LIN {X 0,Y 60.656,Z 289.694,A -85,B 0,C 180,E1 -29046.277,E2 -29046.277} C_VEL
LIN {X 0,Y 62.988,Z 293.733,A -85,B 0,C 180,E1 -29049.53,E2 -29049.53} C_VEL
LIN {X 0,Y 65.947,Z 299.714,A -85,B 0,C 180,E1 -29053.566,E2 -29053.566} C_VEL
LIN {X 0,Y 68.573,Z 306.402,A -85,B 0,C 180,E1 -29057.552,E2 -29057.552} C_VEL
LIN {X 0,Y 68.698,Z 316.329,A -85,B 0,C 180,E1 -29061.954,E2 -29061.954} C_VEL
LIN {X 0,Y 68.38,Z 324.783,A -85,B 0,C 180,E1 -29066.316,E2 -29066.316} C_VEL
LIN {X 0,Y 68.151,Z 327.44,A -85,B 0,C 180,E1 -29067.783,E2 -29067.783} C_VEL
LIN {X 0,Y 64.616,Z 337.01,A -85,B 0,C 180,E1 -29073.116,E2 -29073.116} C_VEL
LIN {X 0,Y 63.028,Z 340.879,A -85,B 0,C 180,E1 -29075.888,E2 -29075.888} C_VEL
LIN {X 0,Y 60.689,Z 345.121,A -85,B 0,C 180,E1 -29079.055,E2 -29079.055} C_VEL
LIN {X 0,Y 55.431,Z 351.353,A -85,B 0,C 180,E1 -29084.685,E2 -29084.685} C_VEL
LIN {X 0,Y 50.566,Z 356.775,A -85,B 0,C 180,E1 -29092.091,E2 -29092.091} C_VEL
LIN {X 0,Y 49.027,Z 359.751,A -85,B 0,C 180,E1 -29097.765,E2 -29097.765} C_VEL
LIN {X 0,Y 48.568,Z 364.973,A -85,B 0,C 180,E1 -29109.693,E2 -29109.693} C_VEL
LIN {X 0,Y 49.872,Z 368.756,A -85,B 0,C 180,E1 -29120.809,E2 -29120.809} C_VEL
LIN {X 0,Y 51.424,Z 370.545,A -85,B 0,C 180,E1 -29126.86,E2 -29126.86} C_VEL
LIN {X 0,Y 56.208,Z 373.025,A -85,B 0,C 180,E1 -29137.968,E2 -29137.968} C_VEL
LIN {X 0,Y 62.698,Z 374.277,A -85,B 0,C 180,E1 -29147.044,E2 -29147.044} C_VEL
LIN {X 0,Y 70.609,Z 374.345,A -85,B 0,C 180,E1 -29154.464,E2 -29154.464} C_VEL
LIN {X 0,Y 78.89,Z 373.239,A -85,B 0,C 180,E1 -29159.999,E2 -29159.999} C_VEL
LIN {X 0,Y 88.109,Z 370.772,A -85,B 0,C 180,E1 -29164.575,E2 -29164.575} C_VEL
LIN {X 0,Y 94.619,Z 368.411,A -85,B 0,C 180,E1 -29167.103,E2 -29167.103} C_VEL
LIN {X 0,Y 97.441,Z 367.133,A -85,B 0,C 180,E1 -29168.293,E2 -29168.293} C_VEL
LIN {X 0,Y 98.808,Z 366.47,A -85,B 0,C 180,E1 -29172.32,E2 -29172.32} C_VEL
LIN {X 0,Y 99.22,Z 366.449,A -85,B 0,C 180,E1 -29176.459,E2 -29176.459} C_VEL
LIN {X 0,Y 99.233,Z 366.885,A -85,B 0,C 180,E1 -29180.739,E2 -29180.739} C_VEL
LIN {X 0,Y 99.149,Z 367.25,A -85,B 0,C 180,E1 -29182.858,E2 -29182.858} C_VEL
LIN {X 0,Y 98.38,Z 367.841,A -85,B 0,C 180,E1 -29184.381,E2 -29184.381} C_VEL
LIN {X 0,Y 90.661,Z 371.366,A -85,B 0,C 180,E1 -29186.942,E2 -29186.942} C_VEL
LIN {X 0,Y 81.683,Z 374.499,A -85,B 0,C 180,E1 -29190.64,E2 -29190.64} C_VEL
LIN {X 0,Y 76.041,Z 376.045,A -85,B 0,C 180,E1 -29193.715,E2 -29193.715} C_VEL
LIN {X 0,Y 70.723,Z 377.095,A -85,B 0,C 180,E1 -29197.346,E2 -29197.346} C_VEL
LIN {X 0,Y 61.158,Z 377.8,A -85,B 0,C 180,E1 -29206.411,E2 -29206.411} C_VEL
LIN {X 0,Y 57.103,Z 377.566,A -85,B 0,C 180,E1 -29212.021,E2 -29212.021} C_VEL
LIN {X 0,Y 53.866,Z 376.846,A -85,B 0,C 180,E1 -29218.542,E2 -29218.542} C_VEL
LIN {X 0,Y 51.484,Z 375.644,A -85,B 0,C 180,E1 -29225.826,E2 -29225.826} C_VEL
LIN {X 0,Y 49.582,Z 373.048,A -85,B 0,C 180,E1 -29237.726,E2 -29237.726} C_VEL
LIN {X 0,Y 49.718,Z 369.258,A -85,B 0,C 180,E1 -29250.001,E2 -29250.001} C_VEL
LIN {X 0,Y 50.679,Z 363.659,A -85,B 0,C 180,E1 -29262.082,E2 -29262.082} C_VEL
LIN {X 0,Y 52.64,Z 359.148,A -85,B 0,C 180,E1 -29269.5,E2 -29269.5} C_VEL
LIN {X 0,Y 55.776,Z 353.792,A -85,B 0,C 180,E1 -29276.17,E2 -29276.17} C_VEL
LIN {X 0,Y 60.052,Z 347.523,A -85,B 0,C 180,E1 -29281.78,E2 -29281.78} C_VEL
LIN {X 0,Y 64.173,Z 342.283,A -85,B 0,C 180,E1 -29285.098,E2 -29285.098} C_VEL
LIN {X 0,Y 68.246,Z 337.731,A -85,B 0,C 180,E1 -29286.999,E2 -29286.999} C_VEL
LIN {X 0,Y 73.162,Z 342.61,A -85,B 0,C 180,E1 -29294.895,E2 -29294.895} C_VEL
LIN {X 0,Y 72.154,Z 341.482,A -85,B 0,C 180,E1 -29297.015,E2 -29297.015} C_VEL
LIN {X 0,Y 65.005,Z 332.075,A -85,B 0,C 180,E1 -29307.278,E2 -29307.278} C_VEL
LIN {X 0,Y 60.672,Z 322.126,A -85,B 0,C 180,E1 -29317.929,E2 -29317.929} C_VEL
LIN {X 0,Y 58.653,Z 313.599,A -85,B 0,C 180,E1 -29326.135,E2 -29326.135} C_VEL
LIN {X 0,Y 57.356,Z 304.126,A -85,B 0,C 180,E1 -29333.846,E2 -29333.846} C_VEL
LIN {X 0,Y 56.745,Z 292.437,A -85,B 0,C 180,E1 -29341.777,E2 -29341.777} C_VEL
LIN {X 0,Y 56.696,Z 289.467,A -85,B 0,C 180,E1 -29343.558,E2 -29343.558} C_VEL
LIN {X 0,Y 55.101,Z 283.817,A -85,B 0,C 180,E1 -29345.813,E2 -29345.813} C_VEL
LIN {X 0,Y 51.561,Z 285.724,A -85,B 0,C 180,E1 -29373.041,E2 -29373.041} C_VEL
LIN {X 0,Y 52.226,Z 286.714,A -85,B 0,C 180,E1 -29382.289,E2 -29382.289} C_VEL
LIN {X 0,Y 52.707,Z 287.689,A -85,B 0,C 180,E1 -29388.185,E2 -29388.185} C_VEL
LIN {X 0,Y 53.227,Z 289.168,A -85,B 0,C 180,E1 -29394.871,E2 -29394.871} C_VEL
LIN {X 0,Y 53.44,Z 290.095,A -85,B 0,C 180,E1 -29397.987,E2 -29397.987} C_VEL
LIN {X 0,Y 56.844,Z 295.639,A -85,B 0,C 180,E1 -29404.195,E2 -29404.195} C_VEL
LIN {X 0,Y 59.186,Z 300.064,A -85,B 0,C 180,E1 -29408.171,E2 -29408.171} C_VEL
LIN {X 0,Y 61.616,Z 305.81,A -85,B 0,C 180,E1 -29412.574,E2 -29412.574} C_VEL
LIN {X 0,Y 62.723,Z 310.076,A -85,B 0,C 180,E1 -29415.395,E2 -29415.395} C_VEL
LIN {X 0,Y 62.547,Z 317.346,A -85,B 0,C 180,E1 -29418.982,E2 -29418.982} C_VEL
LIN {X 0,Y 62,Z 325.309,A -85,B 0,C 180,E1 -29423.49,E2 -29423.49} C_VEL
LIN {X 0,Y 61.705,Z 327.967,A -85,B 0,C 180,E1 -29425.099,E2 -29425.099} C_VEL
LIN {X 0,Y 57.658,Z 338.002,A -85,B 0,C 180,E1 -29431.271,E2 -29431.271} C_VEL
LIN {X 0,Y 54.497,Z 345.164,A -85,B 0,C 180,E1 -29437.408,E2 -29437.408} C_VEL
LIN {X 0,Y 52.168,Z 350.731,A -85,B 0,C 180,E1 -29443.635,E2 -29443.635} C_VEL
LIN {X 0,Y 49.771,Z 356.978,A -85,B 0,C 180,E1 -29452.848,E2 -29452.848} C_VEL
LIN {X 0,Y 49.027,Z 359.751,A -85,B 0,C 180,E1 -29457.765,E2 -29457.765} C_VEL
LIN {X 0,Y 47.9,Z 362.53,A -85,B 0,C 180,E1 -29463.819,E2 -29463.819} C_VEL
LIN {X 0,Y 45.359,Z 366.458,A -85,B 0,C 180,E1 -29474.592,E2 -29474.592} C_VEL
LIN {X 0,Y 44.558,Z 369.668,A -85,B 0,C 180,E1 -29486.581,E2 -29486.581} C_VEL
LIN {X 0,Y 46.096,Z 371.224,A -85,B 0,C 180,E1 -29493.552,E2 -29493.552} C_VEL
LIN {X 0,Y 51.558,Z 373.469,A -85,B 0,C 180,E1 -29504.179,E2 -29504.179} C_VEL
LIN {X 0,Y 59.02,Z 374.707,A -85,B 0,C 180,E1 -29513.16,E2 -29513.16} C_VEL
LIN {X 0,Y 67.483,Z 374.779,A -85,B 0,C 180,E1 -29519.999,E2 -29519.999} C_VEL
LIN {X 0,Y 77.69,Z 373.447,A -85,B 0,C 180,E1 -29525.689,E2 -29525.689} C_VEL
LIN {X 0,Y 86.636,Z 371.138,A -85,B 0,C 180,E1 -29529.337,E2 -29529.337} C_VEL
LIN {X 0,Y 91.606,Z 369.51,A -85,B 0,C 180,E1 -29531.057,E2 -29531.057} C_VEL
LIN {X 0,Y 92.332,Z 369.276,A -85,B 0,C 180,E1 -29533.2,E2 -29533.2} C_VEL
LIN {X 0,Y 92.644,Z 369.375,A -85,B 0,C 180,E1 -29537.664,E2 -29537.664} C_VEL
LIN {X 0,Y 92.666,Z 369.734,A -85,B 0,C 180,E1 -29541.079,E2 -29541.079} C_VEL
LIN {X 0,Y 90.886,Z 370.534,A -85,B 0,C 180,E1 -29541.886,E2 -29541.886} C_VEL
LIN {X 0,Y 84.501,Z 372.83,A -85,B 0,C 180,E1 -29543.813,E2 -29543.813} C_VEL
LIN {X 0,Y 78.302,Z 374.597,A -85,B 0,C 180,E1 -29546.164,E2 -29546.164} C_VEL
LIN {X 0,Y 71.767,Z 376.041,A -85,B 0,C 180,E1 -29549.316,E2 -29549.316} C_VEL
LIN {X 0,Y 66.637,Z 376.892,A -85,B 0,C 180,E1 -29552.465,E2 -29552.465} C_VEL
LIN {X 0,Y 61.218,Z 377.348,A -85,B 0,C 180,E1 -29556.525,E2 -29556.525} C_VEL
LIN {X 0,Y 51.689,Z 376.906,A -85,B 0,C 180,E1 -29567.171,E2 -29567.171} C_VEL
LIN {X 0,Y 47.955,Z 376.122,A -85,B 0,C 180,E1 -29574.113,E2 -29574.113} C_VEL
LIN {X 0,Y 45.12,Z 374.817,A -85,B 0,C 180,E1 -29582.143,E2 -29582.143} C_VEL
LIN {X 0,Y 42.726,Z 372.012,A -85,B 0,C 180,E1 -29595.717,E2 -29595.717} C_VEL
LIN {X 0,Y 42.728,Z 367.921,A -85,B 0,C 180,E1 -29610.002,E2 -29610.002} C_VEL
LIN {X 0,Y 43.489,Z 363.217,A -85,B 0,C 180,E1 -29621.656,E2 -29621.656} C_VEL
LIN {X 0,Y 45.489,Z 358.662,A -85,B 0,C 180,E1 -29630.344,E2 -29630.344} C_VEL
LIN {X 0,Y 48.748,Z 353.283,A -85,B 0,C 180,E1 -29637.942,E2 -29637.942} C_VEL
LIN {X 0,Y 53.154,Z 346.965,A -85,B 0,C 180,E1 -29644.191,E2 -29644.191} C_VEL
LIN {X 0,Y 57.268,Z 341.647,A -85,B 0,C 180,E1 -29647.852,E2 -29647.852} C_VEL
LIN {X 0,Y 63.326,Z 334.785,A -85,B 0,C 180,E1 -29650.695,E2 -29650.695} C_VEL
LIN {X 0,Y 64.269,Z 333.998,A -85,B 0,C 180,E1 -29651.006,E2 -29651.006} C_VEL
LIN {X 0,Y 65.947,Z 335.721,A -85,B 0,C 180,E1 -29653.846,E2 -29653.846} C_VEL
LIN {X 0,Y 65.682,Z 335.325,A -85,B 0,C 180,E1 -29655.933,E2 -29655.933} C_VEL
LIN {X 0,Y 59.31,Z 326.435,A -85,B 0,C 180,E1 -29665.729,E2 -29665.729} C_VEL
LIN {X 0,Y 54.783,Z 315.648,A -85,B 0,C 180,E1 -29677.366,E2 -29677.366} C_VEL
LIN {X 0,Y 52.495,Z 305.883,A -85,B 0,C 180,E1 -29686.451,E2 -29686.451} C_VEL
LIN {X 0,Y 51.074,Z 294.206,A -85,B 0,C 180,E1 -29695.562,E2 -29695.562} C_VEL
LIN {X 0,Y 50.552,Z 287.818,A -85,B 0,C 180,E1 -29699.814,E2 -29699.814} C_VEL
LIN {X 0,Y 49.256,Z 288.07,A -85,B 0,C 180,E1 -29702.789,E2 -29702.789} C_VEL
LIN {X 0,Y 47.867,Z 288.142,A -85,B 0,C 180,E1 -29708.444,E2 -29708.444} C_VEL
LIN {X 0,Y 45.408,Z 289.144,A -85,B 0,C 180,E1 -29727.668,E2 -29727.668} C_VEL
LIN {X 0,Y 45.864,Z 290.076,A -85,B 0,C 180,E1 -29739.985,E2 -29739.985} C_VEL
LIN {X 0,Y 46.261,Z 290.699,A -85,B 0,C 180,E1 -29744.254,E2 -29744.254} C_VEL
LIN {X 0,Y 50.156,Z 296.105,A -85,B 0,C 180,E1 -29755.337,E2 -29755.337} C_VEL
LIN {X 0,Y 52.782,Z 300.941,A -85,B 0,C 180,E1 -29761.564,E2 -29761.564} C_VEL
LIN {X 0,Y 54.882,Z 305.591,A -85,B 0,C 180,E1 -29766.324,E2 -29766.324} C_VEL
LIN {X 0,Y 56.845,Z 311.568,A -85,B 0,C 180,E1 -29771.506,E2 -29771.506} C_VEL
LIN {X 0,Y 56.693,Z 317.172,A -85,B 0,C 180,E1 -29774.724,E2 -29774.724} C_VEL
LIN {X 0,Y 55.798,Z 325.713,A -85,B 0,C 180,E1 -29780.026,E2 -29780.026} C_VEL
LIN {X 0,Y 55.399,Z 328.375,A -85,B 0,C 180,E1 -29781.794,E2 -29781.794} C_VEL
LIN {X 0,Y 51.253,Z 337.891,A -85,B 0,C 180,E1 -29788.034,E2 -29788.034} C_VEL
LIN {X 0,Y 47.781,Z 345.111,A -85,B 0,C 180,E1 -29794.754,E2 -29794.754} C_VEL
LIN {X 0,Y 44.64,Z 351.995,A -85,B 0,C 180,E1 -29803.658,E2 -29803.658} C_VEL
LIN {X 0,Y 42.725,Z 356.721,A -85,B 0,C 180,E1 -29811.721,E2 -29811.721} C_VEL
LIN {X 0,Y 41.534,Z 361.487,A -85,B 0,C 180,E1 -29822.213,E2 -29822.213} C_VEL
LIN {X 0,Y 42.198,Z 367.054,A -85,B 0,C 180,E1 -29838.224,E2 -29838.224} C_VEL
LIN {X 0,Y 46.096,Z 371.224,A -85,B 0,C 180,E1 -29853.552,E2 -29853.552} C_VEL
LIN {X 0,Y 48.29,Z 372.602,A -85,B 0,C 180,E1 -29860.024,E2 -29860.024} C_VEL
LIN {X 0,Y 51.691,Z 374.179,A -85,B 0,C 180,E1 -29870.553,E2 -29870.553} C_VEL
LIN {X 0,Y 55.454,Z 374.983,A -85,B 0,C 180,E1 -29877.995,E2 -29877.995} C_VEL
LIN {X 0,Y 60.161,Z 375.355,A -85,B 0,C 180,E1 -29882.976,E2 -29882.976} C_VEL
LIN {X 0,Y 60.955,Z 375.219,A -85,B 0,C 180,E1 -29883.527,E2 -29883.527} C_VEL
LIN {X 0,Y 65.377,Z 375.203,A -85,B 0,C 180,E1 -29886.171,E2 -29886.171} C_VEL
LIN {X 0,Y 75.32,Z 374.072,A -85,B 0,C 180,E1 -29890.755,E2 -29890.755} C_VEL
LIN {X 0,Y 85.635,Z 371.592,A -85,B 0,C 180,E1 -29894.253,E2 -29894.253} C_VEL
LIN {X 0,Y 85.876,Z 371.694,A -85,B 0,C 180,E1 -29897.284,E2 -29897.284} C_VEL
LIN {X 0,Y 84.263,Z 372.328,A -85,B 0,C 180,E1 -29898.669,E2 -29898.669} C_VEL
LIN {X 0,Y 75.439,Z 374.71,A -85,B 0,C 180,E1 -29901.313,E2 -29901.313} C_VEL
LIN {X 0,Y 67.748,Z 376.091,A -85,B 0,C 180,E1 -29904.516,E2 -29904.516} C_VEL
LIN {X 0,Y 57.272,Z 376.972,A -85,B 0,C 180,E1 -29910.798,E2 -29910.798} C_VEL
LIN {X 0,Y 51.801,Z 376.842,A -85,B 0,C 180,E1 -29915.509,E2 -29915.509} C_VEL
LIN {X 0,Y 46.732,Z 376.239,A -85,B 0,C 180,E1 -29921.242,E2 -29921.242} C_VEL
LIN {X 0,Y 39.006,Z 373.905,A -85,B 0,C 180,E1 -29937.282,E2 -29937.282} C_VEL
LIN {X 0,Y 35.976,Z 370.838,A -85,B 0,C 180,E1 -29952.962,E2 -29952.962} C_VEL
LIN {X 0,Y 35.64,Z 367.71,A -85,B 0,C 180,E1 -29966.033,E2 -29966.033} C_VEL
LIN {X 0,Y 36.068,Z 363.76,A -85,B 0,C 180,E1 -29978.405,E2 -29978.405} C_VEL
LIN {X 0,Y 38.371,Z 358.101,A -85,B 0,C 180,E1 -29991.491,E2 -29991.491} C_VEL
LIN {X 0,Y 41.753,Z 352.703,A -85,B 0,C 180,E1 -30000.331,E2 -30000.331} C_VEL
LIN {X 0,Y 46.404,Z 346.397,A -85,B 0,C 180,E1 -30007.289,E2 -30007.289} C_VEL
LIN {X 0,Y 52.226,Z 339.019,A -85,B 0,C 180,E1 -30012.289,E2 -30012.289} C_VEL
LIN {X 0,Y 57.605,Z 332.868,A -85,B 0,C 180,E1 -30014.55,E2 -30014.55} C_VEL
LIN {X 0,Y 56.453,Z 330.766,A -85,B 0,C 180,E1 -30016.678,E2 -30016.678} C_VEL
LIN {X 0,Y 52.154,Z 324.769,A -85,B 0,C 180,E1 -30023.955,E2 -30023.955} C_VEL
LIN {X 0,Y 48.918,Z 317.846,A -85,B 0,C 180,E1 -30032.166,E2 -30032.166} C_VEL
LIN {X 0,Y 45.801,Z 307.984,A -85,B 0,C 180,E1 -30043.853,E2 -30043.853} C_VEL
LIN {X 0,Y 44.549,Z 300.435,A -85,B 0,C 180,E1 -30052.352,E2 -30052.352} C_VEL
LIN {X 0,Y 44.056,Z 292.312,A -85,B 0,C 180,E1 -30060.001,E2 -30060.001} C_VEL
LIN {X 0,Y 41.977,Z 293.31,A -85,B 0,C 180,E1 -30070.858,E2 -30070.858} C_VEL
LIN {X 0,Y 43.566,Z 296.843,A -85,B 0,C 180,E1 -30100.188,E2 -30100.188} C_VEL
LIN {X 0,Y 44.842,Z 298.788,A -85,B 0,C 180,E1 -30105.65,E2 -30105.65} C_VEL
LIN {X 0,Y 46.781,Z 302.035,A -85,B 0,C 180,E1 -30112.618,E2 -30112.618} C_VEL
LIN {X 0,Y 48.332,Z 305.194,A -85,B 0,C 180,E1 -30117.525,E2 -30117.525} C_VEL
LIN {X 0,Y 50.142,Z 310.246,A -85,B 0,C 180,E1 -30123.619,E2 -30123.619} C_VEL
LIN {X 0,Y 51.378,Z 314.797,A -85,B 0,C 180,E1 -30128.116,E2 -30128.116} C_VEL
LIN {X 0,Y 50.081,Z 324.77,A -85,B 0,C 180,E1 -30134.743,E2 -30134.743} C_VEL
LIN {X 0,Y 49.358,Z 328.727,A -85,B 0,C 180,E1 -30137.666,E2 -30137.666} C_VEL
LIN {X 0,Y 44.759,Z 338.261,A -85,B 0,C 180,E1 -30144.367,E2 -30144.367} C_VEL
LIN {X 0,Y 40.717,Z 345.934,A -85,B 0,C 180,E1 -30152.472,E2 -30152.472} C_VEL
LIN {X 0,Y 37.883,Z 351.526,A -85,B 0,C 180,E1 -30160.69,E2 -30160.69} C_VEL
LIN {X 0,Y 35.252,Z 357.773,A -85,B 0,C 180,E1 -30173.497,E2 -30173.497} C_VEL
LIN {X 0,Y 34.369,Z 362.918,A -85,B 0,C 180,E1 -30187.838,E2 -30187.838} C_VEL
LIN {X 0,Y 35.83,Z 367.54,A -85,B 0,C 180,E1 -30203.951,E2 -30203.951} C_VEL
LIN {X 0,Y 40.549,Z 371.45,A -85,B 0,C 180,E1 -30219.717,E2 -30219.717} C_VEL
LIN {X 0,Y 49.49,Z 374.29,A -85,B 0,C 180,E1 -30233.741,E2 -30233.741} C_VEL
LIN {X 0,Y 56.223,Z 375.144,A -85,B 0,C 180,E1 -30240.108,E2 -30240.108} C_VEL
LIN {X 0,Y 60.955,Z 375.219,A -85,B 0,C 180,E1 -30243.527,E2 -30243.527} C_VEL
LIN {X 0,Y 61.98,Z 375.344,A -85,B 0,C 180,E1 -30244.923,E2 -30244.923} C_VEL
LIN {X 0,Y 62.164,Z 375.496,A -85,B 0,C 180,E1 -30247.783,E2 -30247.783} C_VEL
LIN {X 0,Y 61.331,Z 375.705,A -85,B 0,C 180,E1 -30250.504,E2 -30250.504} C_VEL
LIN {X 0,Y 59.242,Z 375.995,A -85,B 0,C 180,E1 -30254.418,E2 -30254.418} C_VEL
LIN {X 0,Y 54.375,Z 376.362,A -85,B 0,C 180,E1 -30260.889,E2 -30260.889} C_VEL
LIN {X 0,Y 49.622,Z 376.367,A -85,B 0,C 180,E1 -30266.667,E2 -30266.667} C_VEL
LIN {X 0,Y 46.055,Z 376.041,A -85,B 0,C 180,E1 -30270.298,E2 -30270.298} C_VEL
LIN {X 0,Y 37.402,Z 374.413,A -85,B 0,C 180,E1 -30281.271,E2 -30281.271} C_VEL
LIN {X 0,Y 33.277,Z 372.857,A -85,B 0,C 180,E1 -30290.687,E2 -30290.687} C_VEL
LIN {X 0,Y 29.355,Z 369.592,A -85,B 0,C 180,E1 -30308.956,E2 -30308.956} C_VEL
LIN {X 0,Y 28.687,Z 366.448,A -85,B 0,C 180,E1 -30324.365,E2 -30324.365} C_VEL
LIN {X 0,Y 28.958,Z 363.204,A -85,B 0,C 180,E1 -30336.972,E2 -30336.972} C_VEL
LIN {X 0,Y 31.291,Z 357.531,A -85,B 0,C 180,E1 -30353.147,E2 -30353.147} C_VEL
LIN {X 0,Y 34.91,Z 352.09,A -85,B 0,C 180,E1 -30363.618,E2 -30363.618} C_VEL
LIN {X 0,Y 39.853,Z 345.723,A -85,B 0,C 180,E1 -30371.402,E2 -30371.402} C_VEL
LIN {X 0,Y 45.09,Z 339.312,A -85,B 0,C 180,E1 -30376.13,E2 -30376.13} C_VEL
LIN {X 0,Y 49.379,Z 334.319,A -85,B 0,C 180,E1 -30378.352,E2 -30378.352} C_VEL
LIN {X 0,Y 49.142,Z 332.965,A -85,B 0,C 180,E1 -30379.675,E2 -30379.675} C_VEL
LIN {X 0,Y 44.561,Z 324.532,A -85,B 0,C 180,E1 -30391.762,E2 -30391.762} C_VEL
LIN {X 0,Y 42.289,Z 316.472,A -85,B 0,C 180,E1 -30403.093,E2 -30403.093} C_VEL
LIN {X 0,Y 41.242,Z 305.871,A -85,B 0,C 180,E1 -30417.254,E2 -30417.254} C_VEL
LIN {X 0,Y 41.563,Z 299.586,A -85,B 0,C 180,E1 -30423.931,E2 -30423.931} C_VEL
LIN {X 0,Y 40.327,Z 302.748,A -85,B 0,C 180,E1 -30452.764,E2 -30452.764} C_VEL
LIN {X 0,Y 41.45,Z 303.781,A -85,B 0,C 180,E1 -30459.779,E2 -30459.779} C_VEL
LIN {X 0,Y 42.688,Z 306.394,A -85,B 0,C 180,E1 -30466.741,E2 -30466.741} C_VEL
LIN {X 0,Y 44.342,Z 310.984,A -85,B 0,C 180,E1 -30475.093,E2 -30475.093} C_VEL
LIN {X 0,Y 45.632,Z 315.909,A -85,B 0,C 180,E1 -30481.666,E2 -30481.666} C_VEL
LIN {X 0,Y 45.846,Z 317.946,A -85,B 0,C 180,E1 -30483.972,E2 -30483.972} C_VEL
LIN {X 0,Y 44.342,Z 325.739,A -85,B 0,C 180,E1 -30489.773,E2 -30489.773} C_VEL
LIN {X 0,Y 43.599,Z 328.954,A -85,B 0,C 180,E1 -30492.406,E2 -30492.406} C_VEL
LIN {X 0,Y 38.514,Z 338.546,A -85,B 0,C 180,E1 -30499.484,E2 -30499.484} C_VEL
LIN {X 0,Y 34.488,Z 345.439,A -85,B 0,C 180,E1 -30507.329,E2 -30507.329} C_VEL
LIN {X 0,Y 30.38,Z 352.689,A -85,B 0,C 180,E1 -30519.989,E2 -30519.989} C_VEL
LIN {X 0,Y 28.169,Z 357.547,A -85,B 0,C 180,E1 -30532.277,E2 -30532.277} C_VEL
LIN {X 0,Y 27.345,Z 362.591,A -85,B 0,C 180,E1 -30549.551,E2 -30549.551} C_VEL
LIN {X 0,Y 28.775,Z 366.536,A -85,B 0,C 180,E1 -30565.803,E2 -30565.803} C_VEL
LIN {X 0,Y 33.197,Z 370.312,A -85,B 0,C 180,E1 -30582.296,E2 -30582.296} C_VEL
LIN {X 0,Y 36.222,Z 371.879,A -85,B 0,C 180,E1 -30588.811,E2 -30588.811} C_VEL
LIN {X 0,Y 44.608,Z 374.326,A -85,B 0,C 180,E1 -30599.999,E2 -30599.999} C_VEL
LIN {X 0,Y 49.326,Z 375.172,A -85,B 0,C 180,E1 -30604.173,E2 -30604.173} C_VEL
LIN {X 0,Y 57.243,Z 375.756,A -85,B 0,C 180,E1 -30609.36,E2 -30609.36} C_VEL
LIN {X 0,Y 64.919,Z 375.61,A -85,B 0,C 180,E1 -30613.015,E2 -30613.015} C_VEL
LIN {X 0,Y 73.155,Z 374.723,A -85,B 0,C 180,E1 -30616.119,E2 -30616.119} C_VEL
LIN {X 0,Y 64.297,Z 376.02,A -85,B 0,C 180,E1 -30619.142,E2 -30619.142} C_VEL
LIN {X 0,Y 53.978,Z 376.487,A -85,B 0,C 180,E1 -30624.302,E2 -30624.302} C_VEL
LIN {X 0,Y 46.055,Z 376.041,A -85,B 0,C 180,E1 -30630.298,E2 -30630.298} C_VEL
LIN {X 0,Y 41.113,Z 375.367,A -85,B 0,C 180,E1 -30634.435,E2 -30634.435} C_VEL
LIN {X 0,Y 32.639,Z 373.213,A -85,B 0,C 180,E1 -30641.744,E2 -30641.744} C_VEL
LIN {X 0,Y 25.282,Z 370.118,A -85,B 0,C 180,E1 -30653.562,E2 -30653.562} C_VEL
LIN {X 0,Y 22.644,Z 367.929,A -85,B 0,C 180,E1 -30665.206,E2 -30665.206} C_VEL
LIN {X 0,Y 21.81,Z 363.617,A -85,B 0,C 180,E1 -30690.003,E2 -30690.003} C_VEL
LIN {X 0,Y 24.241,Z 356.882,A -85,B 0,C 180,E1 -30715.781,E2 -30715.781} C_VEL
LIN {X 0,Y 28.252,Z 351.429,A -85,B 0,C 180,E1 -30728.458,E2 -30728.458} C_VEL
LIN {X 0,Y 33.604,Z 345.046,A -85,B 0,C 180,E1 -30737.056,E2 -30737.056} C_VEL
LIN {X 0,Y 39.101,Z 338.56,A -85,B 0,C 180,E1 -30741.849,E2 -30741.849} C_VEL
LIN {X 0,Y 41.672,Z 335.549,A -85,B 0,C 180,E1 -30743.238,E2 -30743.238} C_VEL
LIN {X 0,Y 41.657,Z 334.341,A -85,B 0,C 180,E1 -30744.748,E2 -30744.748} C_VEL
LIN {X 0,Y 38.632,Z 326.25,A -85,B 0,C 180,E1 -30758.665,E2 -30758.665} C_VEL
LIN {X 0,Y 37.686,Z 316.568,A -85,B 0,C 180,E1 -30774.651,E2 -30774.651} C_VEL
LIN {X 0,Y 38.523,Z 308.122,A -85,B 0,C 180,E1 -30786.635,E2 -30786.635} C_VEL
LIN {X 0,Y 38.668,Z 307.215,A -85,B 0,C 180,E1 -30787.66,E2 -30787.66} C_VEL
LIN {X 0,Y 37.606,Z 308.192,A -85,B 0,C 180,E1 -30800.859,E2 -30800.859} C_VEL
LIN {X 0,Y 38.642,Z 310.181,A -85,B 0,C 180,E1 -30817.546,E2 -30817.546} C_VEL
LIN {X 0,Y 39.452,Z 312.982,A -85,B 0,C 180,E1 -30825.445,E2 -30825.445} C_VEL
LIN {X 0,Y 40.236,Z 316.519,A -85,B 0,C 180,E1 -30832.229,E2 -30832.229} C_VEL
LIN {X 0,Y 40.561,Z 319.108,A -85,B 0,C 180,E1 -30836.38,E2 -30836.38} C_VEL
LIN {X 0,Y 40.56,Z 320.99,A -85,B 0,C 180,E1 -30838.677,E2 -30838.677} C_VEL
LIN {X 0,Y 38.286,Z 329.224,A -85,B 0,C 180,E1 -30845.662,E2 -30845.662} C_VEL
LIN {X 0,Y 32.671,Z 338.781,A -85,B 0,C 180,E1 -30852.793,E2 -30852.793} C_VEL
LIN {X 0,Y 26.89,Z 347.445,A -85,B 0,C 180,E1 -30864.349,E2 -30864.349} C_VEL
LIN {X 0,Y 22.795,Z 353.8,A -85,B 0,C 180,E1 -30878.865,E2 -30878.865} C_VEL
LIN {X 0,Y 20.356,Z 359.842,A -85,B 0,C 180,E1 -30901.187,E2 -30901.187} C_VEL
LIN {X 0,Y 21.378,Z 364.95,A -85,B 0,C 180,E1 -30926.373,E2 -30926.373} C_VEL
LIN {X 0,Y 25.036,Z 368.435,A -85,B 0,C 180,E1 -30943.695,E2 -30943.695} C_VEL
LIN {X 0,Y 33.05,Z 372.296,A -85,B 0,C 180,E1 -30959.999,E2 -30959.999} C_VEL
LIN {X 0,Y 42.757,Z 374.748,A -85,B 0,C 180,E1 -30969.527,E2 -30969.527} C_VEL
LIN {X 0,Y 52.931,Z 375.976,A -85,B 0,C 180,E1 -30975.399,E2 -30975.399} C_VEL
LIN {X 0,Y 51.462,Z 376.003,A -85,B 0,C 180,E1 -30977.07,E2 -30977.07} C_VEL
LIN {X 0,Y 38.871,Z 374.819,A -85,B 0,C 180,E1 -30985.314,E2 -30985.314} C_VEL
LIN {X 0,Y 33.159,Z 373.534,A -85,B 0,C 180,E1 -30992.031,E2 -30992.031} C_VEL
LIN {X 0,Y 26.044,Z 370.833,A -85,B 0,C 180,E1 -31007.579,E2 -31007.579} C_VEL
LIN {X 0,Y 22.644,Z 367.929,A -85,B 0,C 180,E1 -31025.206,E2 -31025.206} C_VEL
LIN {X 0,Y 21.548,Z 366.349,A -85,B 0,C 180,E1 -31034.059,E2 -31034.059} C_VEL
LIN {X 0,Y 19.852,Z 363.604,A -85,B 0,C 180,E1 -31047.721,E2 -31047.721} C_VEL
LIN {X 0,Y 18.66,Z 360.341,A -85,B 0,C 180,E1 -31062.366,E2 -31062.366} C_VEL
LIN {X 0,Y 19.484,Z 354.318,A -85,B 0,C 180,E1 -31086.719,E2 -31086.719} C_VEL
LIN {X 0,Y 22.22,Z 350.371,A -85,B 0,C 180,E1 -31096.834,E2 -31096.834} C_VEL
LIN {X 0,Y 27.853,Z 344.264,A -85,B 0,C 180,E1 -31105.094,E2 -31105.094} C_VEL
LIN {X 0,Y 33.724,Z 337.649,A -85,B 0,C 180,E1 -31109.478,E2 -31109.478} C_VEL
LIN {X 0,Y 34.666,Z 336.584,A -85,B 0,C 180,E1 -31109.889,E2 -31109.889} C_VEL
LIN {X 0,Y 33.71,Z 332.371,A -85,B 0,C 180,E1 -31118.603,E2 -31118.603} C_VEL
LIN {X 0,Y 33.41,Z 324.071,A -85,B 0,C 180,E1 -31135.477,E2 -31135.477} C_VEL
LIN {X 0,Y 35.372,Z 314.699,A -85,B 0,C 180,E1 -31151.462,E2 -31151.462} C_VEL
LIN {X 0,Y 34.906,Z 315.165,A -85,B 0,C 180,E1 -31163.748,E2 -31163.748} C_VEL
LIN {X 0,Y 35.551,Z 316.806,A -85,B 0,C 180,E1 -31176.377,E2 -31176.377} C_VEL
LIN {X 0,Y 35.778,Z 319.245,A -85,B 0,C 180,E1 -31183.443,E2 -31183.443} C_VEL
LIN {X 0,Y 35.882,Z 321.983,A -85,B 0,C 180,E1 -31189.11,E2 -31189.11} C_VEL
LIN {X 0,Y 35.82,Z 323.506,A -85,B 0,C 180,E1 -31191.523,E2 -31191.523} C_VEL
LIN {X 0,Y 33.427,Z 329.817,A -85,B 0,C 180,E1 -31197.249,E2 -31197.249} C_VEL
LIN {X 0,Y 26.566,Z 340.077,A -85,B 0,C 180,E1 -31204.537,E2 -31204.537} C_VEL
LIN {X 0,Y 20.738,Z 347.654,A -85,B 0,C 180,E1 -31215.263,E2 -31215.263} C_VEL
LIN {X 0,Y 16.379,Z 353.221,A -85,B 0,C 180,E1 -31229.996,E2 -31229.996} C_VEL
LIN {X 0,Y 13.721,Z 357.721,A -85,B 0,C 180,E1 -31250.892,E2 -31250.892} C_VEL
LIN {X 0,Y 14.333,Z 363.466,A -85,B 0,C 180,E1 -31290.634,E2 -31290.634} C_VEL
LIN {X 0,Y 17.84,Z 366.693,A -85,B 0,C 180,E1 -31310.009,E2 -31310.009} C_VEL
LIN {X 0,Y 24.737,Z 370.295,A -85,B 0,C 180,E1 -31325.594,E2 -31325.594} C_VEL
LIN {X 0,Y 33.936,Z 373.368,A -85,B 0,C 180,E1 -31334.973,E2 -31334.973} C_VEL
LIN {X 0,Y 30.011,Z 372.585,A -85,B 0,C 180,E1 -31340.496,E2 -31340.496} C_VEL
LIN {X 0,Y 21.393,Z 369.58,A -85,B 0,C 180,E1 -31354.788,E2 -31354.788} C_VEL
LIN {X 0,Y 15.655,Z 365.452,A -85,B 0,C 180,E1 -31383.329,E2 -31383.329} C_VEL
LIN {X 0,Y 14.855,Z 361.948,A -85,B 0,C 180,E1 -31410.004,E2 -31410.004} C_VEL
LIN {X 0,Y 17.292,Z 356.218,A -85,B 0,C 180,E1 -31440.538,E2 -31440.538} C_VEL
LIN {X 0,Y 22.22,Z 350.371,A -85,B 0,C 180,E1 -31456.834,E2 -31456.834} C_VEL
LIN {X 0,Y 24.329,Z 347.663,A -85,B 0,C 180,E1 -31462.028,E2 -31462.028} C_VEL
LIN {X 0,Y 26.33,Z 343.614,A -85,B 0,C 180,E1 -31469.181,E2 -31469.181} C_VEL
LIN {X 0,Y 27.629,Z 339.507,A -85,B 0,C 180,E1 -31476.792,E2 -31476.792} C_VEL
LIN {X 0,Y 28.234,Z 335.602,A -85,B 0,C 180,E1 -31484.896,E2 -31484.896} C_VEL
LIN {X 0,Y 28.294,Z 334.715,A -85,B 0,C 180,E1 -31487.105,E2 -31487.105} C_VEL
LIN {X 0,Y 30.526,Z 324.869,A -85,B 0,C 180,E1 -31509.945,E2 -31509.945} C_VEL
LIN {X 0,Y 31.955,Z 321.339,A -85,B 0,C 180,E1 -31516.588,E2 -31516.588} C_VEL
LIN {X 0,Y 31.735,Z 322.123,A -85,B 0,C 180,E1 -31527.64,E2 -31527.64} C_VEL
LIN {X 0,Y 31.932,Z 323.72,A -85,B 0,C 180,E1 -31536.609,E2 -31536.609} C_VEL
LIN {X 0,Y 31.626,Z 325.781,A -85,B 0,C 180,E1 -31541.812,E2 -31541.812} C_VEL
LIN {X 0,Y 30.049,Z 329.325,A -85,B 0,C 180,E1 -31545.437,E2 -31545.437} C_VEL
LIN {X 0,Y 27.908,Z 332.806,A -85,B 0,C 180,E1 -31547.153,E2 -31547.153} C_VEL
LIN {X 0,Y 21.399,Z 341.261,A -85,B 0,C 180,E1 -31551.842,E2 -31551.842} C_VEL
LIN {X 0,Y 14.559,Z 348.781,A -85,B 0,C 180,E1 -31561.131,E2 -31561.131} C_VEL
LIN {X 0,Y 7.71,Z 355.908,A -85,B 0,C 180,E1 -31589.992,E2 -31589.992} C_VEL
LIN {X 0,Y 8.616,Z 362.856,A -85,B 0,C 180,E1 -31672.228,E2 -31672.228} C_VEL
LIN {X 0,Y 16.424,Z 367.457,A -85,B 0,C 180,E1 -31695.795,E2 -31695.795} C_VEL
LIN {X 0,Y 15.214,Z 367.034,A -85,B 0,C 180,E1 -31702.505,E2 -31702.505} C_VEL
LIN {X 0,Y 8.099,Z 361.452,A -85,B 0,C 180,E1 -31754.694,E2 -31754.694} C_VEL
LIN {X 0,Y 9.529,Z 356.766,A -85,B 0,C 180,E1 -31803.591,E2 -31803.591} C_VEL
LIN {X 0,Y 14.742,Z 351.453,A -85,B 0,C 180,E1 -31826.552,E2 -31826.552} C_VEL
LIN {X 0,Y 21.206,Z 345.219,A -85,B 0,C 180,E1 -31835.705,E2 -31835.705} C_VEL
LIN {X 0,Y 28.389,Z 337.591,A -85,B 0,C 180,E1 -31839.474,E2 -31839.474} C_VEL
LIN {X 0,Y 28.294,Z 334.715,A -85,B 0,C 180,E1 -31847.105,E2 -31847.105} C_VEL
LIN {X 0,Y 27.902,Z 333.778,A -85,B 0,C 180,E1 -31851.287,E2 -31851.287} C_VEL
LIN {X 0,Y 25.429,Z 333.13,A -85,B 0,C 180,E1 -31868.708,E2 -31868.708} C_VEL
LIN {X 0,Y 25.721,Z 332.245,A -85,B 0,C 180,E1 -31872.45,E2 -31872.45} C_VEL
LIN {X 0,Y 28.23,Z 327.868,A -85,B 0,C 180,E1 -31882.246,E2 -31882.246} C_VEL
LIN {X 0,Y 27.959,Z 328.889,A -85,B 0,C 180,E1 -31890.183,E2 -31890.183} C_VEL
LIN {X 0,Y 27.747,Z 329.452,A -85,B 0,C 180,E1 -31891.84,E2 -31891.84} C_VEL
LIN {X 0,Y 26.043,Z 332.203,A -85,B 0,C 180,E1 -31892.667,E2 -31892.667} C_VEL
LIN {X 0,Y 18.789,Z 341.324,A -85,B 0,C 180,E1 -31892.681,E2 -31892.681} C_VEL
LIN {X 0,Y 13.112,Z 347.293,A -85,B 0,C 180,E1 -31892.415,E2 -31892.415} C_VEL
LIN {X 0,Y 6.002,Z 353.553,A -85,B 0,C 180,E1 -31888.556,E2 -31888.556} C_VEL
LIN {X 0,Y 1.456,Z 357.215,A -85,B 0,C 180,E1 -31860.032,E2 -31860.032} C_VEL
LIN {X 0,Y 3.662,Z 356.014,A -85,B 0,C 180,E1 -31843.705,E2 -31843.705} C_VEL
LIN {X 0,Y 10.614,Z 350.636,A -85,B 0,C 180,E1 -31853.383,E2 -31853.383} C_VEL
LIN {X 0,Y 17.664,Z 344.319,A -85,B 0,C 180,E1 -31854.121,E2 -31854.121} C_VEL
LIN {X 0,Y 22.868,Z 339.074,A -85,B 0,C 180,E1 -31853.527,E2 -31853.527} C_VEL
LIN {X 0,Y 23.306,Z 338.046,A -85,B 0,C 180,E1 -31855.678,E2 -31855.678} C_VEL
LIN {X 0,Y 25.721,Z 332.245,A -85,B 0,C 180,E1 -31872.45,E2 -31872.45} C_VEL
LIN {X 0,Y 27.241,Z 333.785,A -85,B 0,C 180,E1 -31878.734,E2 -31878.734} C_VEL
LIN {X 0,Y 27.241,Z 600,A -85,B 0,C 180,E1 -31878.734,E2 -31878.734} C_VEL
LIN {X 0,Y 27.241,Z 600,A -85,B 0,C 180,E1 -31878.734,E2 -31878.734}

QRS_NEXT_CUT()

QRS_NEXT()
QRS_HOME()

END
